TYPE csp_transfer_infeed_accU_waterfallAdjust_enum :
(
	CSP_TRANSFER_INFEED_ACCU_WATERFALL_ADJUST_STATUS_NOT_INITIALIZED 							:=  0,
	CSP_TRANSFER_INFEED_ACCU_WATERFALL_ADJUST_STATUS_DISABLED 									:=  10,
	CSP_TRANSFER_INFEED_ACCU_WATERFALL_ADJUST_STATUS_POSITION_CHECK								:=  20,
	CSP_TRANSFER_INFEED_ACCU_WATERFALL_ADJUST_STATUS_ENABLE_REQUEST 							:=  30,
	CSP_TRANSFER_INFEED_ACCU_WATERFALL_ADJUST_STATUS_ENABLED 									:=  40,
	CSP_TRANSFER_INFEED_ACCU_WATERFALL_ADJUST_STATUS_ABS_MOVE_REQUEST							:= 50,
	CSP_TRANSFER_INFEED_ACCU_WATERFALL_ADJUST_STATUS_ABS_MOVING									:= 60,
	CSP_TRANSFER_INFEED_ACCU_WATERFALL_ADJUST_STATUS_STOP_REQUEST 								:= 70,
	CSP_TRANSFER_INFEED_ACCU_WATERFALL_ADJUST_STATUS_DISABLE_REQUEST 							:= 80,
	CSP_TRANSFER_INFEED_ACCU_WATERFALL_ADJUST_STATUS_DISABLING 									:= 90
) := CSP_TRANSFER_INFEED_ACCU_WATERFALL_ADJUST_STATUS_NOT_INITIALIZED;
END_TYPE

(* stored: Version 1.1.0.1, ProductVersion 3.1.4024.3
   DUT csp_transfer_infeed_accU_waterfallAdjust_enum: Id {90b764a6-771c-4799-838b-2ebfd5352476} *)
